{attribute 'GeneratedUsingTerminal: AT2050-0500-0024'}
{attribute addProperty BoxType "AT2050-0500-0024"}
{attribute addProperty Id "A_0089_AT2050_5501_0018_AT2050_5501AT2050_01D6DEDF80"}
{attribute addProperty CRC "534594657"}
{attribute addProperty Size "80"}
TYPE A_0055_AT2050_0500_0024_1FDD4461 EXTENDS AT2050_86175B41 :
STRUCT
	{attribute addProperty Name "A_0089_AT2050_5501_0018_AT2050_5501"}
	A_0089_AT2050_5501_0018_AT2050_5501 : AT2050_01D6DEDF;
END_STRUCT
END_TYPE

(* stored: Version 1.2.0.0, ProductVersion 3.1.4024.9
   DUT A_0055_AT2050_0500_0024_1FDD4461: Id {6c70f85f-31e3-4da9-9eb2-6a4d9366daba} *)
